Staubli VAL3: eraseField.pgx

program eraseField(num x_nColumn)
  local bool l_bOk
  local num l_nFieldLength
  local string l_sDisplay
begin
  // This program erases an area of the screen where the textBox value
  // should be displayed. The area start at column number passed as parameter
  //
  // Input Param
  // x_nColumn  : Column to start erasing
  //
  //Created 21/12/05                              CCUR
  //--------------------------------------------------------------
  l_sDisplay=" "
  toNum(pw:sTxtBoxLen[nFocused],l_nFieldLength,l_bOk)
  call ut:strAlign(l_sDisplay,l_nFieldLength,"R"," ")
  gotoxy(x_nColumn,nTxtPosY[nFocused])
  put(l_sDisplay)
end
